// TIA Portal V17 export
// export: Created 2024-08-09T12:50:41.9449587Z, ExportSetting WithDefaults, DisplayName Totally Integrated Automation Portal, DisplayVersion V17 Update 7, DisplayName TIA Portal Openness, DisplayVersion V17 Update 7, DisplayName TIA Portal Version Control Interface, DisplayVersion V17, DisplayName STEP 7 Professional, DisplayVersion V17 Update 7, DisplayName STEP 7 Safety, DisplayVersion V17 Update 6, DisplayName WinCC Professional, DisplayVersion V17 Update 7
DATA_BLOCK "Gestion_Erreur_DB"   // DB26
VERSION : 0.1
// stored: AutoNumber true, DBAccessibleFromOPCUA true, DBAccessibleFromWebserver true, InstanceOfName Gestion_Erreur, InstanceOfType FB
"Gestion_Erreur"
   // VAR_INPUT
   //    diResultState : DInt;
   // END_VAR
   // VAR_OUTPUT
   //    erreur : String;
   // END_VAR
   // VAR_IN_OUT
   //    stSql4SiemensInterface : "utSql4SiemensInterface";
   // END_VAR
BEGIN
END_DATA_BLOCK
